(* IEC 61131-3 sources: standardizer-tutorial-lib/src/ControlModules/valves, 4 files *)

(* ---- TypeValveState.st ---- *)
NAMESPACE Simatic.Ax.Tutorial
    TYPE
        ValveState : (Open, Closed, Error, Undefined, HardError) := Undefined;
    END_TYPE
END_NAMESPACE

(* ---- IValve.st ---- *)
NAMESPACE Simatic.Ax.Tutorial
    INTERFACE IValve
        METHOD Open
        END_METHOD
        METHOD Close
        END_METHOD
        METHOD GetState : ValveState
        END_METHOD
    END_INTERFACE
END_NAMESPACE

(* ---- Valve.st ---- *)
USING Simatic.Ax.IO.Output;

NAMESPACE Simatic.Ax.Tutorial.Solution
    CLASS Valve IMPLEMENTS IValve

        VAR PRIVATE
            _valveState : BOOL;
        END_VAR

        VAR PUBLIC
            qValve : IBinOutput;
        END_VAR

        METHOD PUBLIC SetRefToDQ
            VAR_INPUT
                dq : IBinOutput;
            END_VAR
            qValve := dq;
        END_METHOD

        METHOD PUBLIC Close

            IF (qValve <> NULL) THEN
                qValve.SetOff();
            END_IF;
            _valveState := false;
        END_METHOD

        METHOD PUBLIC Open
            IF (qValve <> NULL) THEN
                qValve.SetOn();
            END_IF;
            _valveState := true;
        END_METHOD

        METHOD PUBLIC GetState : ValveState
            IF (_valveState) THEN
                GetState := ValveState#Open;
            ELSE
                GetState := ValveState#Closed;
            END_IF;
        END_METHOD
    END_CLASS

END_NAMESPACE

(* ---- ValveFbClosed.st ---- *)
USING Simatic.Ax.IO.Input;
NAMESPACE Simatic.Ax.Tutorial

    CLASS ValveFbClosed EXTENDS Solution.Valve IMPLEMENTS IValve

        VAR PUBLIC
            signalFbClosed : IBinSignal;
        END_VAR

        // GetState will be overwritten with new functionality
        METHOD PUBLIC OVERRIDE GetState : ValveState
            IF(signalFbClosed <> NULL) THEN
                IF (signalFbClosed.Q()) THEN
                    GetState := ValveState#Closed;
                ELSE
                    GetState := ValveState#Open;
                END_IF;
            ELSE;
                GetState := ValveState#HardError;
            END_IF;
        END_METHOD

    END_CLASS

END_NAMESPACE
